// TIA Portal V20 export
TYPE "typeCmHmiInterfaceBrakeTest"
// stored: Access Published, Namespace Unit1.Em8
   STRUCT
      thicknessAxisZ : "LER_typeBrakeTestEmInterface";
   END_STRUCT;
END_TYPE
